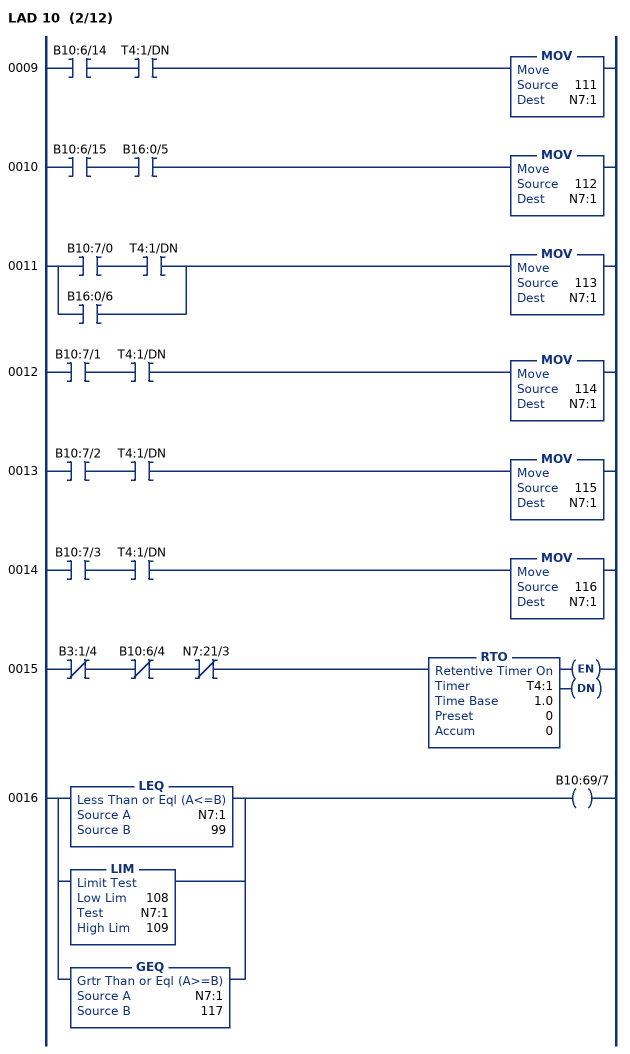
% Rung: 9 %
SOR XIC B10:6/14 XIC T4:1/DN MOV 111 N7:1 EOR
% Rung: 10 %
SOR XIC B10:6/15 XIC B16:0/5 MOV 112 N7:1 EOR
% Rung: 11 %
SOR BST XIC B10:7/0 XIC T4:1/DN NXB XIC B16:0/6 BND MOV 113 N7:1 EOR
% Rung: 12 %
SOR XIC B10:7/1 XIC T4:1/DN MOV 114 N7:1 EOR
% Rung: 13 %
SOR XIC B10:7/2 XIC T4:1/DN MOV 115 N7:1 EOR
% Rung: 14 %
SOR XIC B10:7/3 XIC T4:1/DN MOV 116 N7:1 EOR
% Rung: 15 %
SOR XIO B3:1/4 XIO B10:6/4 XIO N7:21/3 RTO T4:1 1.0 0 0 EOR
% Rung: 16 %
SOR BST LEQ N7:1 99 NXB LIM 108 N7:1 109 NXB GEQ N7:1 117 BND OTE B10:69/7 EOR

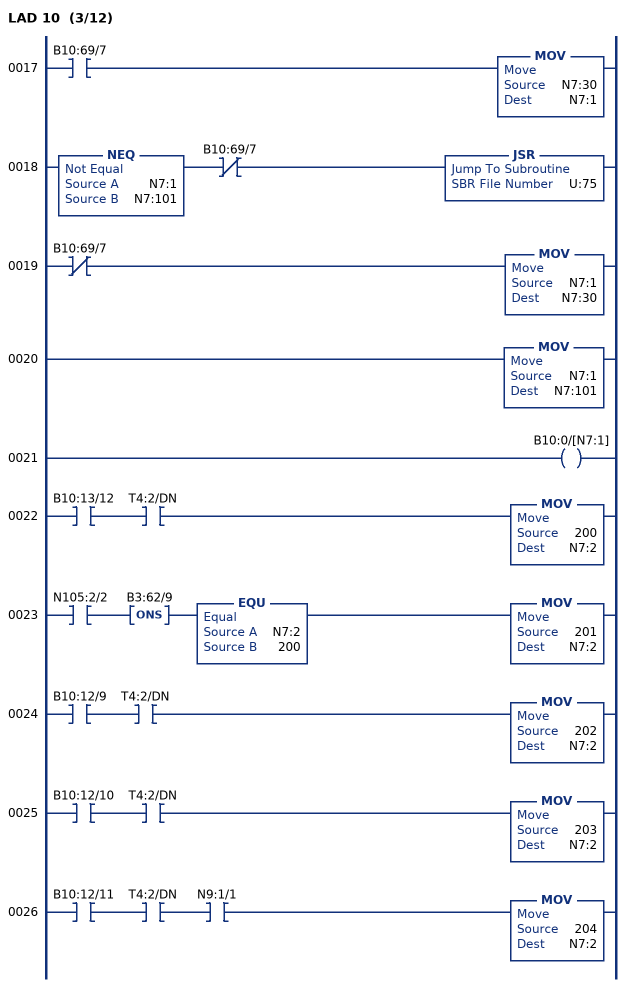
% Rung: 17 %
SOR XIC B10:69/7 MOV N7:30 N7:1 EOR
% Rung: 18 %
SOR NEQ N7:1 N7:101 XIO B10:69/7 JSR U:75 EOR
% Rung: 19 %
SOR XIO B10:69/7 MOV N7:1 N7:30 EOR
% Rung: 20 %
SOR MOV N7:1 N7:101 EOR
% Rung: 21 %
SOR OTE B10:0/[N7:1] EOR
% Rung: 22 %
SOR XIC B10:13/12 XIC T4:2/DN MOV 200 N7:2 EOR
% Rung: 23 %
SOR XIC N105:2/2 OSR B3:62/9 EQU N7:2 200 MOV 201 N7:2 EOR
% Rung: 24 %
SOR XIC B10:12/9 XIC T4:2/DN MOV 202 N7:2 EOR
% Rung: 25 %
SOR XIC B10:12/10 XIC T4:2/DN MOV 203 N7:2 EOR
% Rung: 26 %
SOR XIC B10:12/11 XIC T4:2/DN XIC N9:1/1 MOV 204 N7:2 EOR

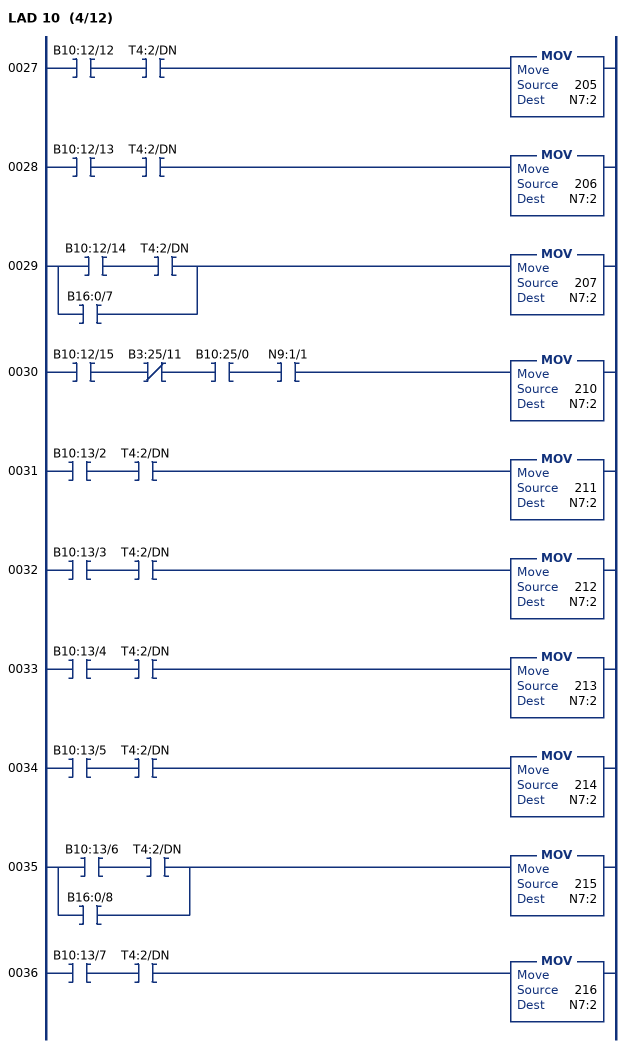
% Rung: 27 %
SOR XIC B10:12/12 XIC T4:2/DN MOV 205 N7:2 EOR
% Rung: 28 %
SOR XIC B10:12/13 XIC T4:2/DN MOV 206 N7:2 EOR
% Rung: 29 %
SOR BST XIC B10:12/14 XIC T4:2/DN NXB XIC B16:0/7 BND MOV 207 N7:2 EOR
% Rung: 30 %
SOR XIC B10:12/15 XIO B3:25/11 XIC B10:25/0 XIC N9:1/1 MOV 210 N7:2 EOR
% Rung: 31 %
SOR XIC B10:13/2 XIC T4:2/DN MOV 211 N7:2 EOR
% Rung: 32 %
SOR XIC B10:13/3 XIC T4:2/DN MOV 212 N7:2 EOR
% Rung: 33 %
SOR XIC B10:13/4 XIC T4:2/DN MOV 213 N7:2 EOR
% Rung: 34 %
SOR XIC B10:13/5 XIC T4:2/DN MOV 214 N7:2 EOR
% Rung: 35 %
SOR BST XIC B10:13/6 XIC T4:2/DN NXB XIC B16:0/8 BND MOV 215 N7:2 EOR
% Rung: 36 %
SOR XIC B10:13/7 XIC T4:2/DN MOV 216 N7:2 EOR

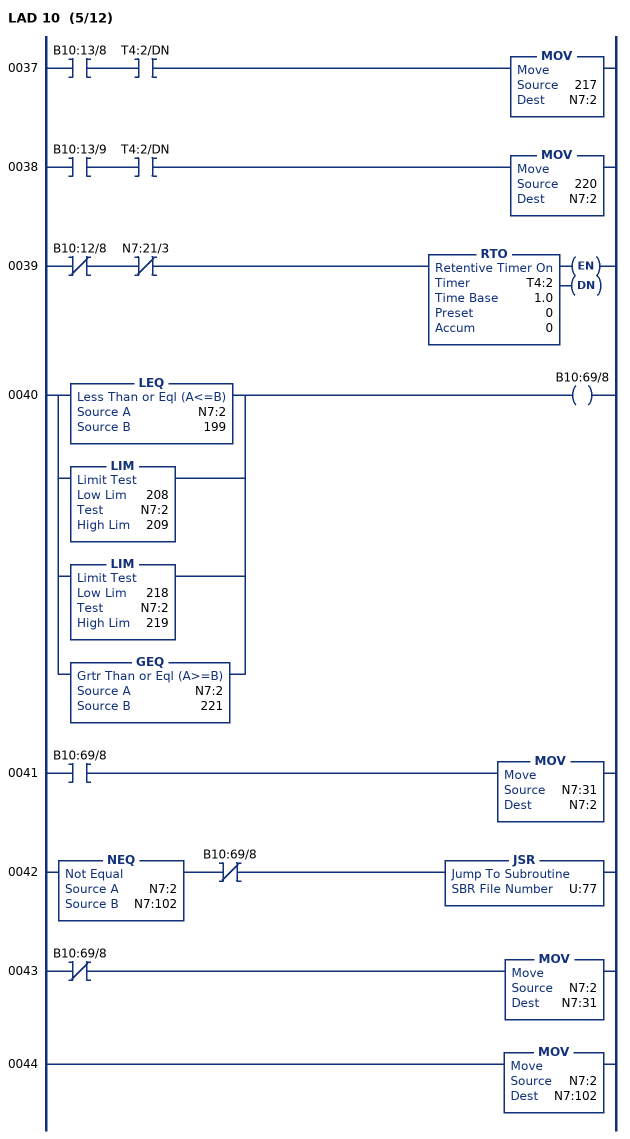
% Rung: 37 %
SOR XIC B10:13/8 XIC T4:2/DN MOV 217 N7:2 EOR
% Rung: 38 %
SOR XIC B10:13/9 XIC T4:2/DN MOV 220 N7:2 EOR
% Rung: 39 %
SOR XIO B10:12/8 XIO N7:21/3 RTO T4:2 1.0 0 0 EOR
% Rung: 40 %
SOR BST LEQ N7:2 199 NXB LIM 208 N7:2 209 NXB LIM 218 N7:2 219 NXB GEQ N7:2 221 BND OTE B10:69/8 EOR
% Rung: 41 %
SOR XIC B10:69/8 MOV N7:31 N7:2 EOR
% Rung: 42 %
SOR NEQ N7:2 N7:102 XIO B10:69/8 JSR U:77 EOR
% Rung: 43 %
SOR XIO B10:69/8 MOV N7:2 N7:31 EOR
% Rung: 44 %
SOR MOV N7:2 N7:102 EOR

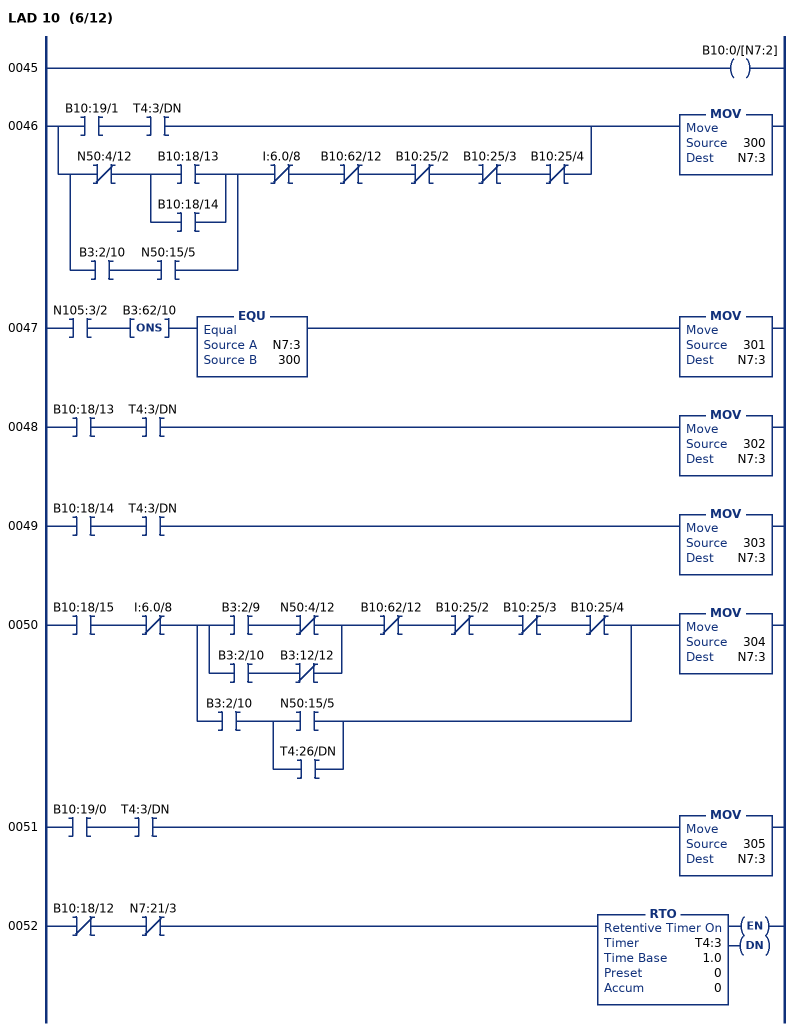
% Rung: 45 %
SOR OTE B10:0/[N7:2] EOR
% Rung: 46 %
SOR BST XIC B10:19/1 XIC T4:3/DN NXB BST XIO N50:4/12 BST XIC B10:18/13 NXB XIC B10:18/14 BND NXB XIC B3:2/10 XIC N50:15/5 BND XIO I:6.0/8 XIO B10:62/12 XIO B10:25/2 XIO B10:25/3 XIO B10:25/4 BND MOV 300 N7:3 EOR
% Rung: 47 %
SOR XIC N105:3/2 OSR B3:62/10 EQU N7:3 300 MOV 301 N7:3 EOR
% Rung: 48 %
SOR XIC B10:18/13 XIC T4:3/DN MOV 302 N7:3 EOR
% Rung: 49 %
SOR XIC B10:18/14 XIC T4:3/DN MOV 303 N7:3 EOR
% Rung: 50 %
SOR XIC B10:18/15 XIO I:6.0/8 BST BST XIC B3:2/9 XIO N50:4/12 NXB XIC B3:2/10 XIO B3:12/12 BND XIO B10:62/12 XIO B10:25/2 XIO B10:25/3 XIO B10:25/4 NXB XIC B3:2/10 BST XIC N50:15/5 NXB XIC T4:26/DN BND BND MOV 304 N7:3 EOR
% Rung: 51 %
SOR XIC B10:19/0 XIC T4:3/DN MOV 305 N7:3 EOR
% Rung: 52 %
SOR XIO B10:18/12 XIO N7:21/3 RTO T4:3 1.0 0 0 EOR

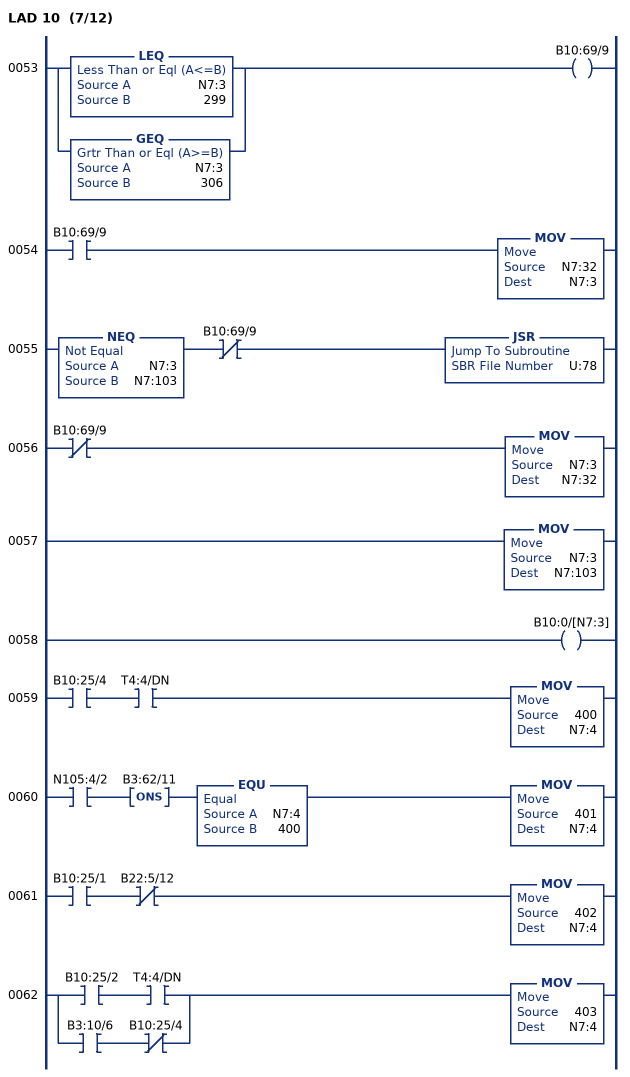
% Rung: 53 %
SOR BST LEQ N7:3 299 NXB GEQ N7:3 306 BND OTE B10:69/9 EOR
% Rung: 54 %
SOR XIC B10:69/9 MOV N7:32 N7:3 EOR
% Rung: 55 %
SOR NEQ N7:3 N7:103 XIO B10:69/9 JSR U:78 EOR
% Rung: 56 %
SOR XIO B10:69/9 MOV N7:3 N7:32 EOR
% Rung: 57 %
SOR MOV N7:3 N7:103 EOR
% Rung: 58 %
SOR OTE B10:0/[N7:3] EOR
% Rung: 59 %
SOR XIC B10:25/4 XIC T4:4/DN MOV 400 N7:4 EOR
% Rung: 60 %
SOR XIC N105:4/2 OSR B3:62/11 EQU N7:4 400 MOV 401 N7:4 EOR
% Rung: 61 %
SOR XIC B10:25/1 XIO B22:5/12 MOV 402 N7:4 EOR
% Rung: 62 %
SOR BST XIC B10:25/2 XIC T4:4/DN NXB XIC B3:10/6 XIO B10:25/4 BND MOV 403 N7:4 EOR

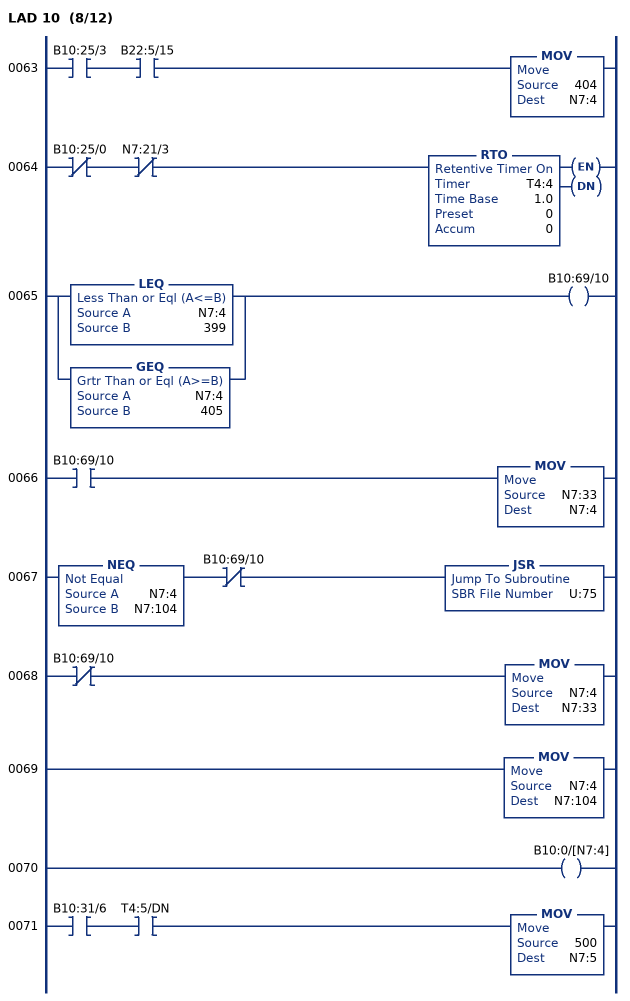
% Rung: 63 %
SOR XIC B10:25/3 XIC B22:5/15 MOV 404 N7:4 EOR
% Rung: 64 %
SOR XIO B10:25/0 XIO N7:21/3 RTO T4:4 1.0 0 0 EOR
% Rung: 65 %
SOR BST LEQ N7:4 399 NXB GEQ N7:4 405 BND OTE B10:69/10 EOR
% Rung: 66 %
SOR XIC B10:69/10 MOV N7:33 N7:4 EOR
% Rung: 67 %
SOR NEQ N7:4 N7:104 XIO B10:69/10 JSR U:75 EOR
% Rung: 68 %
SOR XIO B10:69/10 MOV N7:4 N7:33 EOR
% Rung: 69 %
SOR MOV N7:4 N7:104 EOR
% Rung: 70 %
SOR OTE B10:0/[N7:4] EOR
% Rung: 71 %
SOR XIC B10:31/6 XIC T4:5/DN MOV 500 N7:5 EOR

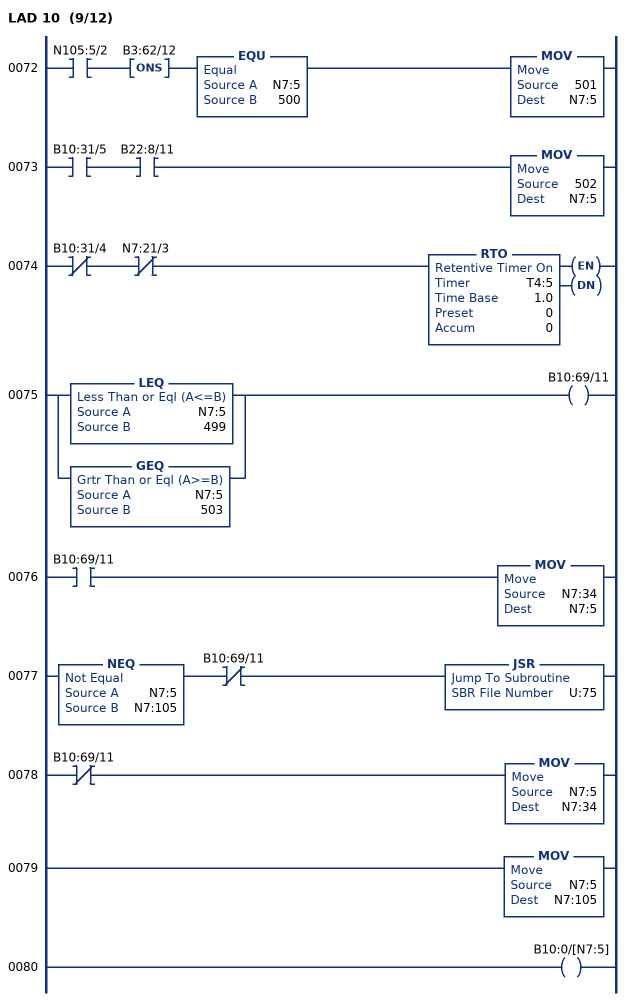
% Rung: 72 %
SOR XIC N105:5/2 OSR B3:62/12 EQU N7:5 500 MOV 501 N7:5 EOR
% Rung: 73 %
SOR XIC B10:31/5 XIC B22:8/11 MOV 502 N7:5 EOR
% Rung: 74 %
SOR XIO B10:31/4 XIO N7:21/3 RTO T4:5 1.0 0 0 EOR
% Rung: 75 %
SOR BST LEQ N7:5 499 NXB GEQ N7:5 503 BND OTE B10:69/11 EOR
% Rung: 76 %
SOR XIC B10:69/11 MOV N7:34 N7:5 EOR
% Rung: 77 %
SOR NEQ N7:5 N7:105 XIO B10:69/11 JSR U:75 EOR
% Rung: 78 %
SOR XIO B10:69/11 MOV N7:5 N7:34 EOR
% Rung: 79 %
SOR MOV N7:5 N7:105 EOR
% Rung: 80 %
SOR OTE B10:0/[N7:5] EOR

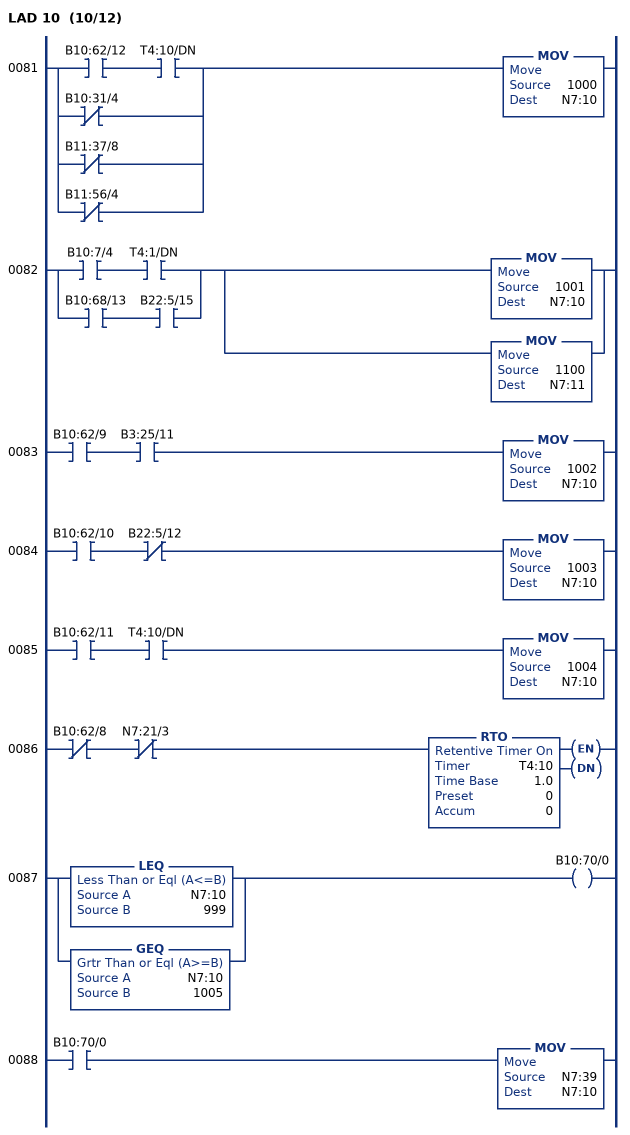
% Rung: 81 %
SOR BST XIC B10:62/12 XIC T4:10/DN NXB XIO B10:31/4 NXB XIO B11:37/8 NXB XIO B11:56/4 BND MOV 1000 N7:10 EOR
% Rung: 82 %
SOR BST XIC B10:7/4 XIC T4:1/DN NXB XIC B10:68/13 XIC B22:5/15 BND BST MOV 1001 N7:10 NXB MOV 1100 N7:11 BND EOR
% Rung: 83 %
SOR XIC B10:62/9 XIC B3:25/11 MOV 1002 N7:10 EOR
% Rung: 84 %
SOR XIC B10:62/10 XIO B22:5/12 MOV 1003 N7:10 EOR
% Rung: 85 %
SOR XIC B10:62/11 XIC T4:10/DN MOV 1004 N7:10 EOR
% Rung: 86 %
SOR XIO B10:62/8 XIO N7:21/3 RTO T4:10 1.0 0 0 EOR
% Rung: 87 %
SOR BST LEQ N7:10 999 NXB GEQ N7:10 1005 BND OTE B10:70/0 EOR
% Rung: 88 %
SOR XIC B10:70/0 MOV N7:39 N7:10 EOR

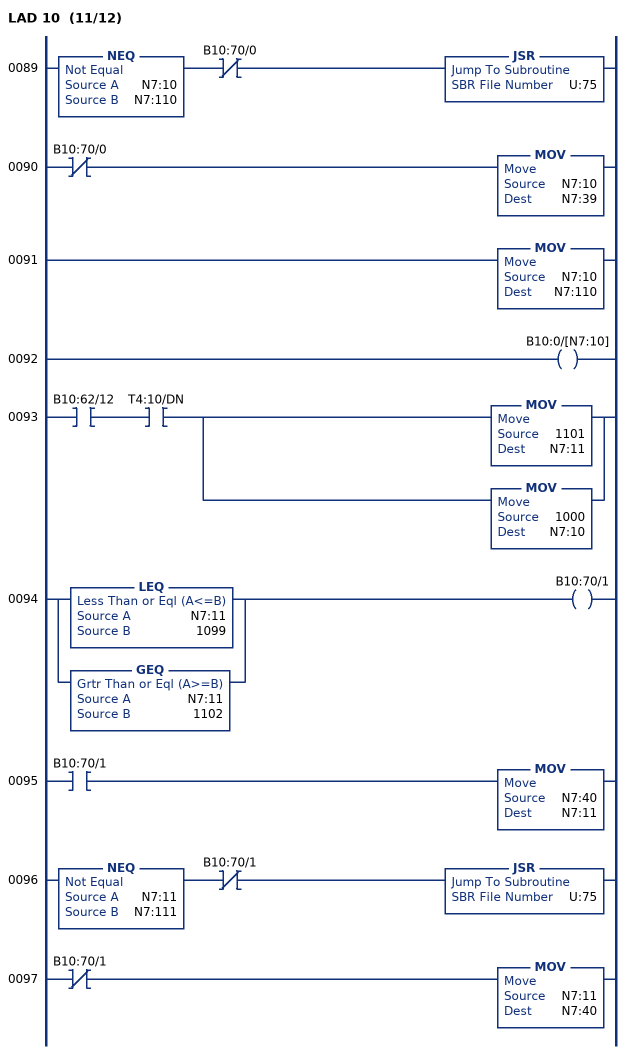
% Rung: 89 %
SOR NEQ N7:10 N7:110 XIO B10:70/0 JSR U:75 EOR
% Rung: 90 %
SOR XIO B10:70/0 MOV N7:10 N7:39 EOR
% Rung: 91 %
SOR MOV N7:10 N7:110 EOR
% Rung: 92 %
SOR OTE B10:0/[N7:10] EOR
% Rung: 93 %
SOR XIC B10:62/12 XIC T4:10/DN BST MOV 1101 N7:11 NXB MOV 1000 N7:10 BND EOR
% Rung: 94 %
SOR BST LEQ N7:11 1099 NXB GEQ N7:11 1102 BND OTE B10:70/1 EOR
% Rung: 95 %
SOR XIC B10:70/1 MOV N7:40 N7:11 EOR
% Rung: 96 %
SOR NEQ N7:11 N7:111 XIO B10:70/1 JSR U:75 EOR
% Rung: 97 %
SOR XIO B10:70/1 MOV N7:11 N7:40 EOR

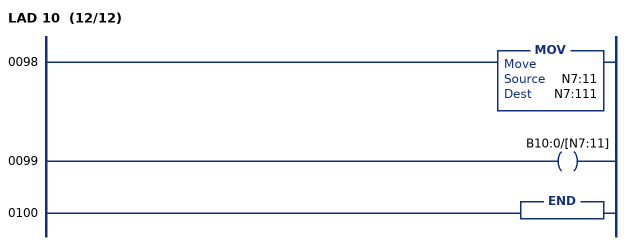
% Rung: 98 %
SOR MOV N7:11 N7:111 EOR
% Rung: 99 %
SOR OTE B10:0/[N7:11] EOR
% Rung: 100 %
SOR END EOR

LADDER 11
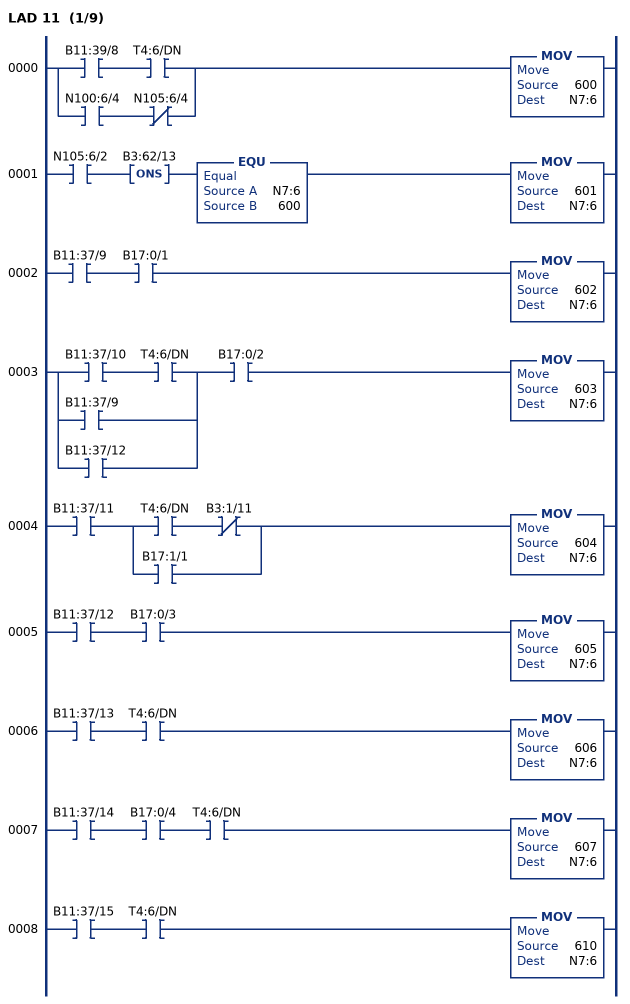
% Rung: 0 %
SOR BST XIC B11:39/8 XIC T4:6/DN NXB XIC N100:6/4 XIO N105:6/4 BND MOV 600 N7:6 EOR
% Rung: 1 %
SOR XIC N105:6/2 OSR B3:62/13 EQU N7:6 600 MOV 601 N7:6 EOR
% Rung: 2 %
SOR XIC B11:37/9 XIC B17:0/1 MOV 602 N7:6 EOR
% Rung: 3 %
SOR BST XIC B11:37/10 XIC T4:6/DN NXB BST XIC B11:37/9 NXB XIC B11:37/12 BND BND XIC B17:0/2 MOV 603 N7:6 EOR
% Rung: 4 %
SOR XIC B11:37/11 BST XIC T4:6/DN XIO B3:1/11 NXB XIC B17:1/1 BND MOV 604 N7:6 EOR
% Rung: 5 %
SOR XIC B11:37/12 XIC B17:0/3 MOV 605 N7:6 EOR
% Rung: 6 %
SOR XIC B11:37/13 XIC T4:6/DN MOV 606 N7:6 EOR
% Rung: 7 %
SOR XIC B11:37/14 XIC B17:0/4 XIC T4:6/DN MOV 607 N7:6 EOR
% Rung: 8 %
SOR XIC B11:37/15 XIC T4:6/DN MOV 610 N7:6 EOR

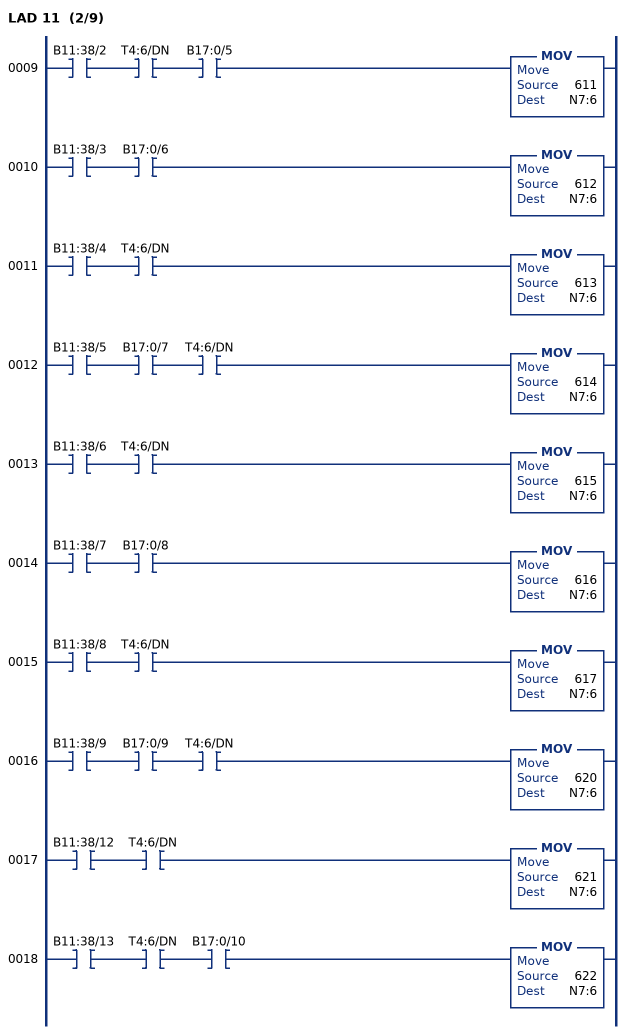
% Rung: 9 %
SOR XIC B11:38/2 XIC T4:6/DN XIC B17:0/5 MOV 611 N7:6 EOR
% Rung: 10 %
SOR XIC B11:38/3 XIC B17:0/6 MOV 612 N7:6 EOR
% Rung: 11 %
SOR XIC B11:38/4 XIC T4:6/DN MOV 613 N7:6 EOR
% Rung: 12 %
SOR XIC B11:38/5 XIC B17:0/7 XIC T4:6/DN MOV 614 N7:6 EOR
% Rung: 13 %
SOR XIC B11:38/6 XIC T4:6/DN MOV 615 N7:6 EOR
% Rung: 14 %
SOR XIC B11:38/7 XIC B17:0/8 MOV 616 N7:6 EOR
% Rung: 15 %
SOR XIC B11:38/8 XIC T4:6/DN MOV 617 N7:6 EOR
% Rung: 16 %
SOR XIC B11:38/9 XIC B17:0/9 XIC T4:6/DN MOV 620 N7:6 EOR
% Rung: 17 %
SOR XIC B11:38/12 XIC T4:6/DN MOV 621 N7:6 EOR
% Rung: 18 %
SOR XIC B11:38/13 XIC T4:6/DN XIC B17:0/10 MOV 622 N7:6 EOR

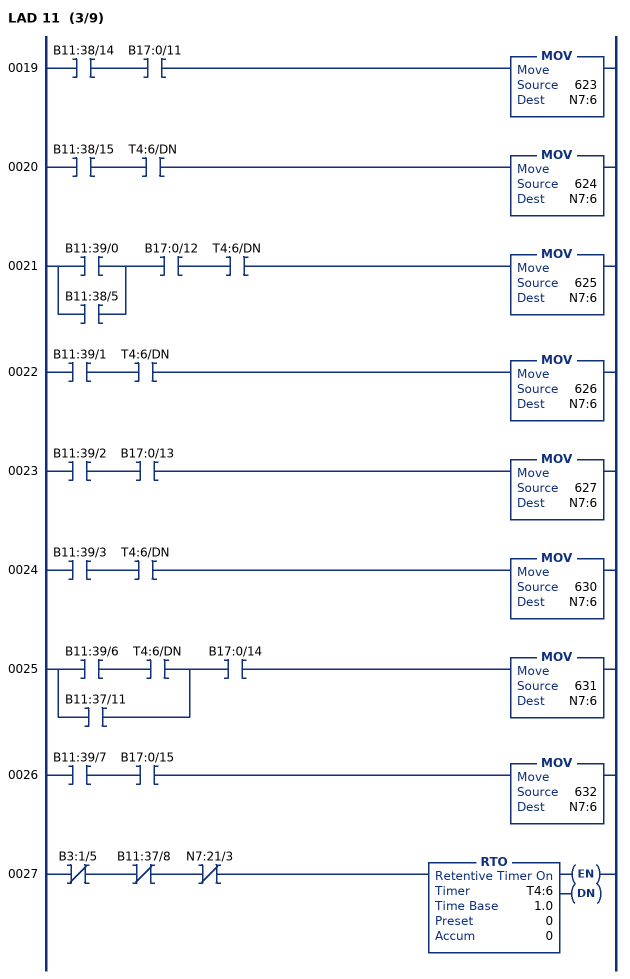
% Rung: 19 %
SOR XIC B11:38/14 XIC B17:0/11 MOV 623 N7:6 EOR
% Rung: 20 %
SOR XIC B11:38/15 XIC T4:6/DN MOV 624 N7:6 EOR
% Rung: 21 %
SOR BST XIC B11:39/0 NXB XIC B11:38/5 BND XIC B17:0/12 XIC T4:6/DN MOV 625 N7:6 EOR
% Rung: 22 %
SOR XIC B11:39/1 XIC T4:6/DN MOV 626 N7:6 EOR
% Rung: 23 %
SOR XIC B11:39/2 XIC B17:0/13 MOV 627 N7:6 EOR
% Rung: 24 %
SOR XIC B11:39/3 XIC T4:6/DN MOV 630 N7:6 EOR
% Rung: 25 %
SOR BST XIC B11:39/6 XIC T4:6/DN NXB XIC B11:37/11 BND XIC B17:0/14 MOV 631 N7:6 EOR
% Rung: 26 %
SOR XIC B11:39/7 XIC B17:0/15 MOV 632 N7:6 EOR
% Rung: 27 %
SOR XIO B3:1/5 XIO B11:37/8 XIO N7:21/3 RTO T4:6 1.0 0 0 EOR

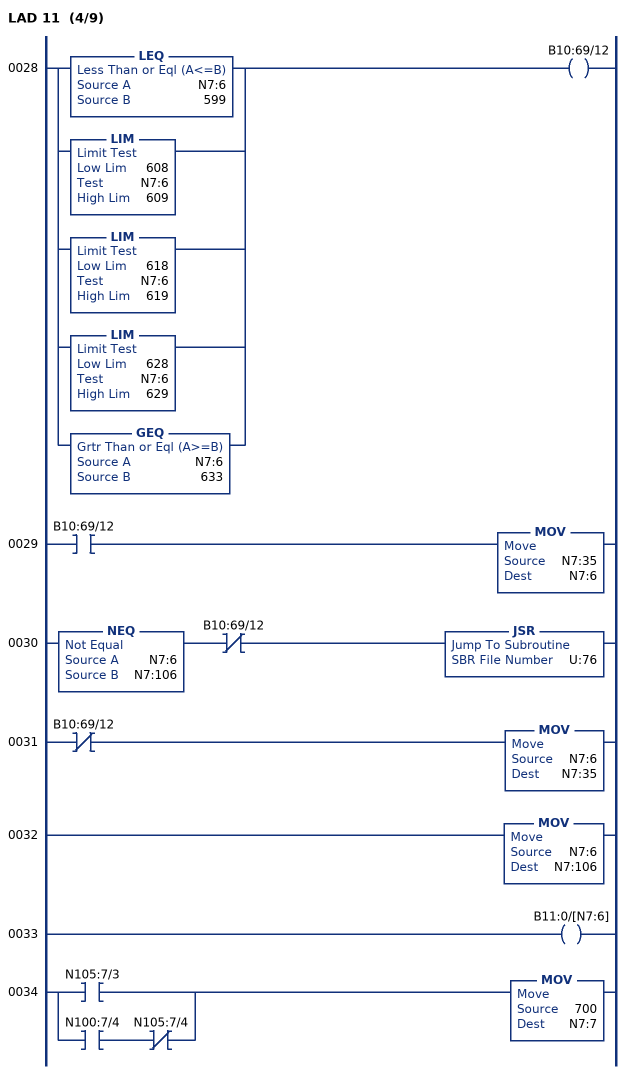
% Rung: 28 %
SOR BST LEQ N7:6 599 NXB LIM 608 N7:6 609 NXB LIM 618 N7:6 619 NXB LIM 628 N7:6 629 NXB GEQ N7:6 633 BND OTE B10:69/12 EOR
% Rung: 29 %
SOR XIC B10:69/12 MOV N7:35 N7:6 EOR
% Rung: 30 %
SOR NEQ N7:6 N7:106 XIO B10:69/12 JSR U:76 EOR
% Rung: 31 %
SOR XIO B10:69/12 MOV N7:6 N7:35 EOR
% Rung: 32 %
SOR MOV N7:6 N7:106 EOR
% Rung: 33 %
SOR OTE B11:0/[N7:6] EOR
% Rung: 34 %
SOR BST XIC N105:7/3 NXB XIC N100:7/4 XIO N105:7/4 BND MOV 700 N7:7 EOR

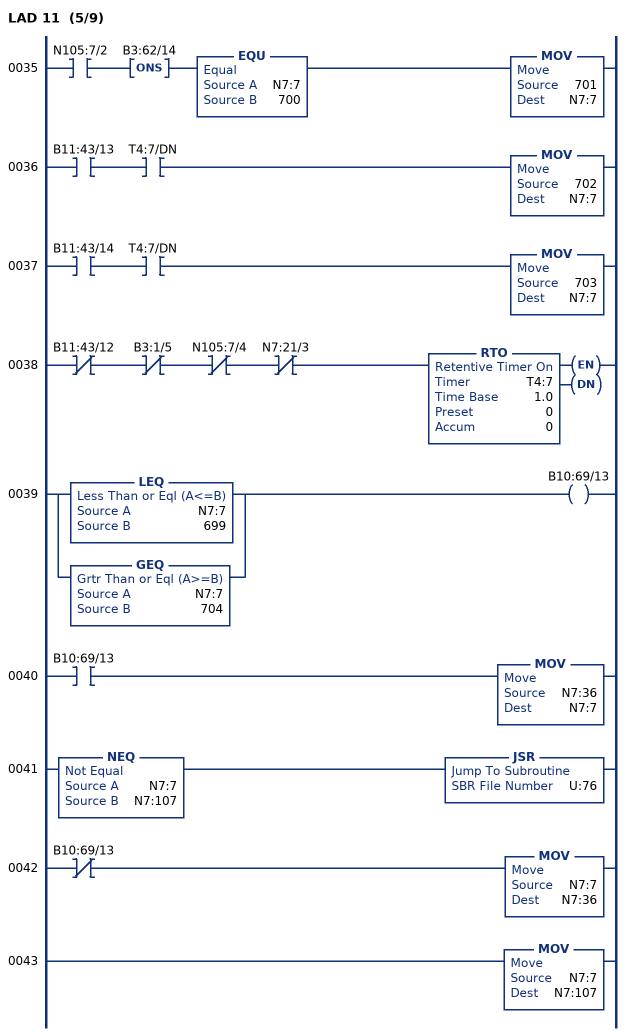
% Rung: 35 %
SOR XIC N105:7/2 OSR B3:62/14 EQU N7:7 700 MOV 701 N7:7 EOR
% Rung: 36 %
SOR XIC B11:43/13 XIC T4:7/DN MOV 702 N7:7 EOR
% Rung: 37 %
SOR XIC B11:43/14 XIC T4:7/DN MOV 703 N7:7 EOR
% Rung: 38 %
SOR XIO B11:43/12 XIO B3:1/5 XIO N105:7/4 XIO N7:21/3 RTO T4:7 1.0 0 0 EOR
% Rung: 39 %
SOR BST LEQ N7:7 699 NXB GEQ N7:7 704 BND OTE B10:69/13 EOR
% Rung: 40 %
SOR XIC B10:69/13 MOV N7:36 N7:7 EOR
% Rung: 41 %
SOR NEQ N7:7 N7:107 JSR U:76 EOR
% Rung: 42 %
SOR XIO B10:69/13 MOV N7:7 N7:36 EOR
% Rung: 43 %
SOR MOV N7:7 N7:107 EOR

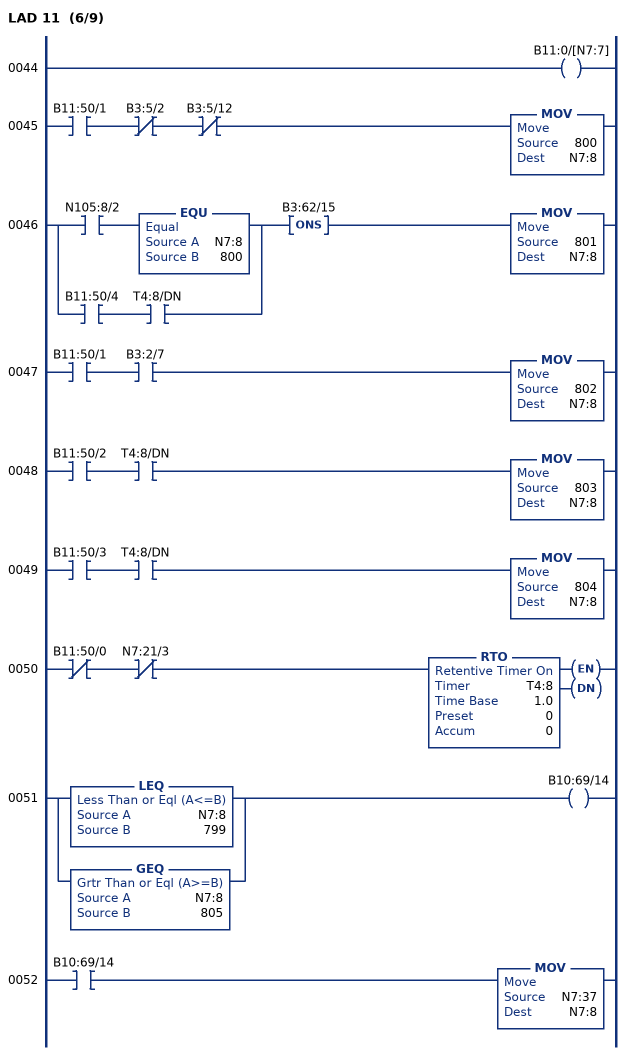
% Rung: 44 %
SOR OTE B11:0/[N7:7] EOR
% Rung: 45 %
SOR XIC B11:50/1 XIO B3:5/2 XIO B3:5/12 MOV 800 N7:8 EOR
% Rung: 46 %
SOR BST XIC N105:8/2 EQU N7:8 800 NXB XIC B11:50/4 XIC T4:8/DN BND OSR B3:62/15 MOV 801 N7:8 EOR
% Rung: 47 %
SOR XIC B11:50/1 XIC B3:2/7 MOV 802 N7:8 EOR
% Rung: 48 %
SOR XIC B11:50/2 XIC T4:8/DN MOV 803 N7:8 EOR
% Rung: 49 %
SOR XIC B11:50/3 XIC T4:8/DN MOV 804 N7:8 EOR
% Rung: 50 %
SOR XIO B11:50/0 XIO N7:21/3 RTO T4:8 1.0 0 0 EOR
% Rung: 51 %
SOR BST LEQ N7:8 799 NXB GEQ N7:8 805 BND OTE B10:69/14 EOR
% Rung: 52 %
SOR XIC B10:69/14 MOV N7:37 N7:8 EOR

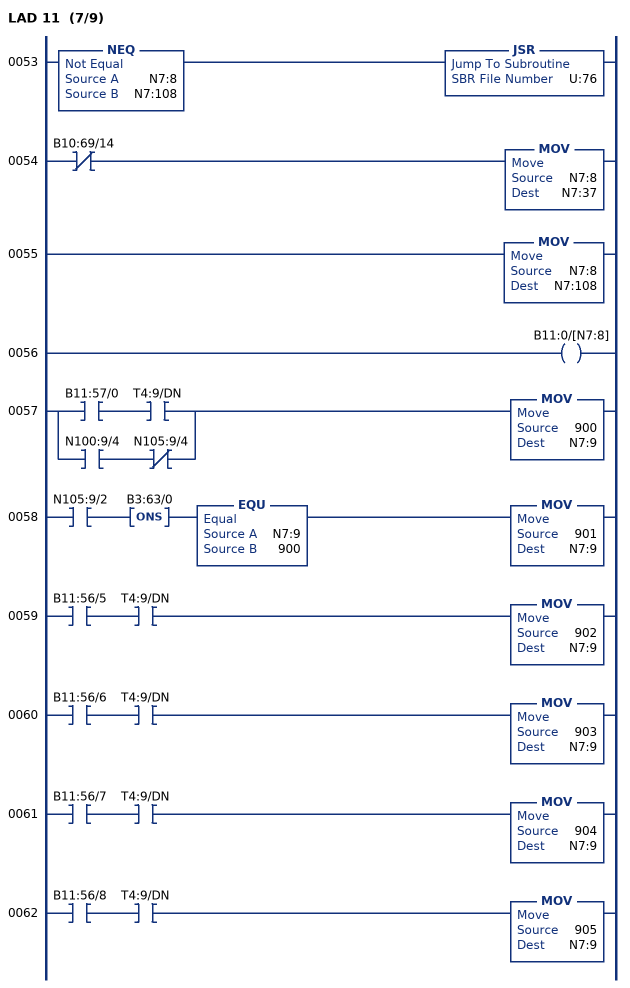
% Rung: 53 %
SOR NEQ N7:8 N7:108 JSR U:76 EOR
% Rung: 54 %
SOR XIO B10:69/14 MOV N7:8 N7:37 EOR
% Rung: 55 %
SOR MOV N7:8 N7:108 EOR
% Rung: 56 %
SOR OTE B11:0/[N7:8] EOR
% Rung: 57 %
SOR BST XIC B11:57/0 XIC T4:9/DN NXB XIC N100:9/4 XIO N105:9/4 BND MOV 900 N7:9 EOR
% Rung: 58 %
SOR XIC N105:9/2 OSR B3:63/0 EQU N7:9 900 MOV 901 N7:9 EOR
% Rung: 59 %
SOR XIC B11:56/5 XIC T4:9/DN MOV 902 N7:9 EOR
% Rung: 60 %
SOR XIC B11:56/6 XIC T4:9/DN MOV 903 N7:9 EOR
% Rung: 61 %
SOR XIC B11:56/7 XIC T4:9/DN MOV 904 N7:9 EOR
% Rung: 62 %
SOR XIC B11:56/8 XIC T4:9/DN MOV 905 N7:9 EOR

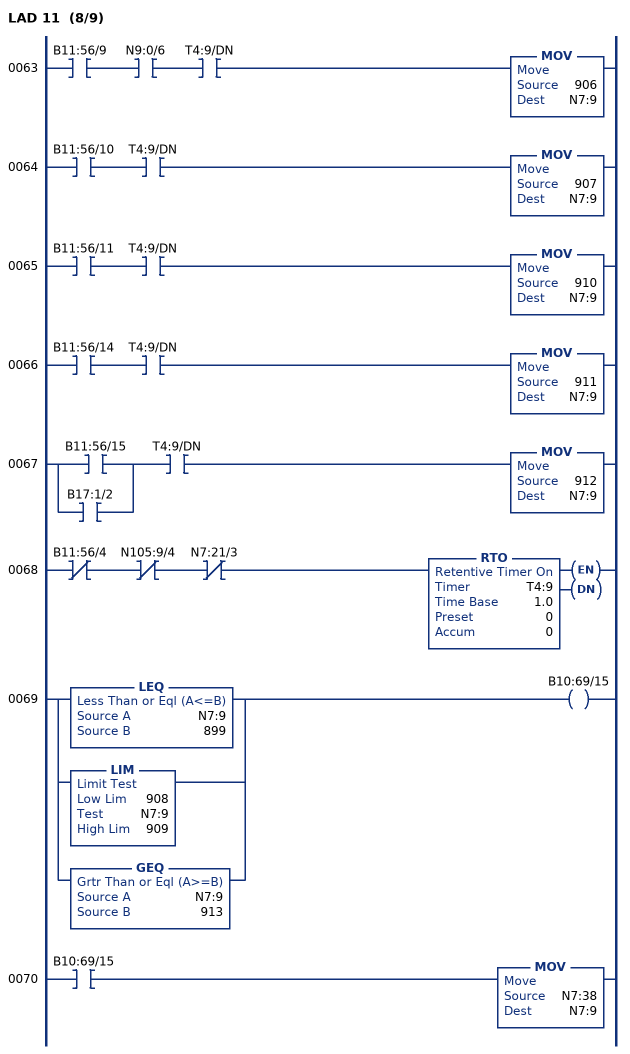
% Rung: 63 %
SOR XIC B11:56/9 XIC N9:0/6 XIC T4:9/DN MOV 906 N7:9 EOR
% Rung: 64 %
SOR XIC B11:56/10 XIC T4:9/DN MOV 907 N7:9 EOR
% Rung: 65 %
SOR XIC B11:56/11 XIC T4:9/DN MOV 910 N7:9 EOR
% Rung: 66 %
SOR XIC B11:56/14 XIC T4:9/DN MOV 911 N7:9 EOR
% Rung: 67 %
SOR BST XIC B11:56/15 NXB XIC B17:1/2 BND XIC T4:9/DN MOV 912 N7:9 EOR
% Rung: 68 %
SOR XIO B11:56/4 XIO N105:9/4 XIO N7:21/3 RTO T4:9 1.0 0 0 EOR
% Rung: 69 %
SOR BST LEQ N7:9 899 NXB LIM 908 N7:9 909 NXB GEQ N7:9 913 BND OTE B10:69/15 EOR
% Rung: 70 %
SOR XIC B10:69/15 MOV N7:38 N7:9 EOR

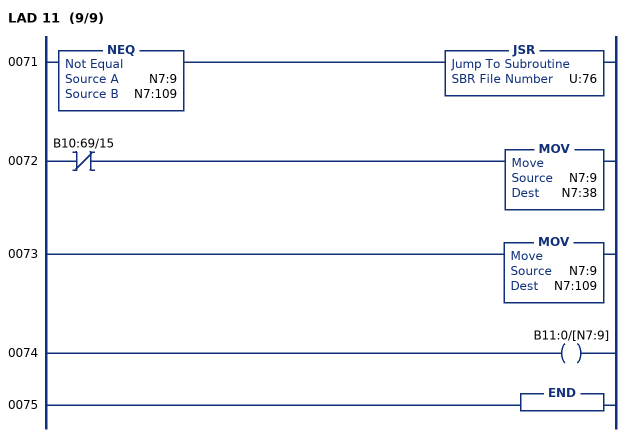
% Rung: 71 %
SOR NEQ N7:9 N7:109 JSR U:76 EOR
% Rung: 72 %
SOR XIO B10:69/15 MOV N7:9 N7:38 EOR
% Rung: 73 %
SOR MOV N7:9 N7:109 EOR
% Rung: 74 %
SOR OTE B11:0/[N7:9] EOR
% Rung: 75 %
SOR END EOR

LADDER 15
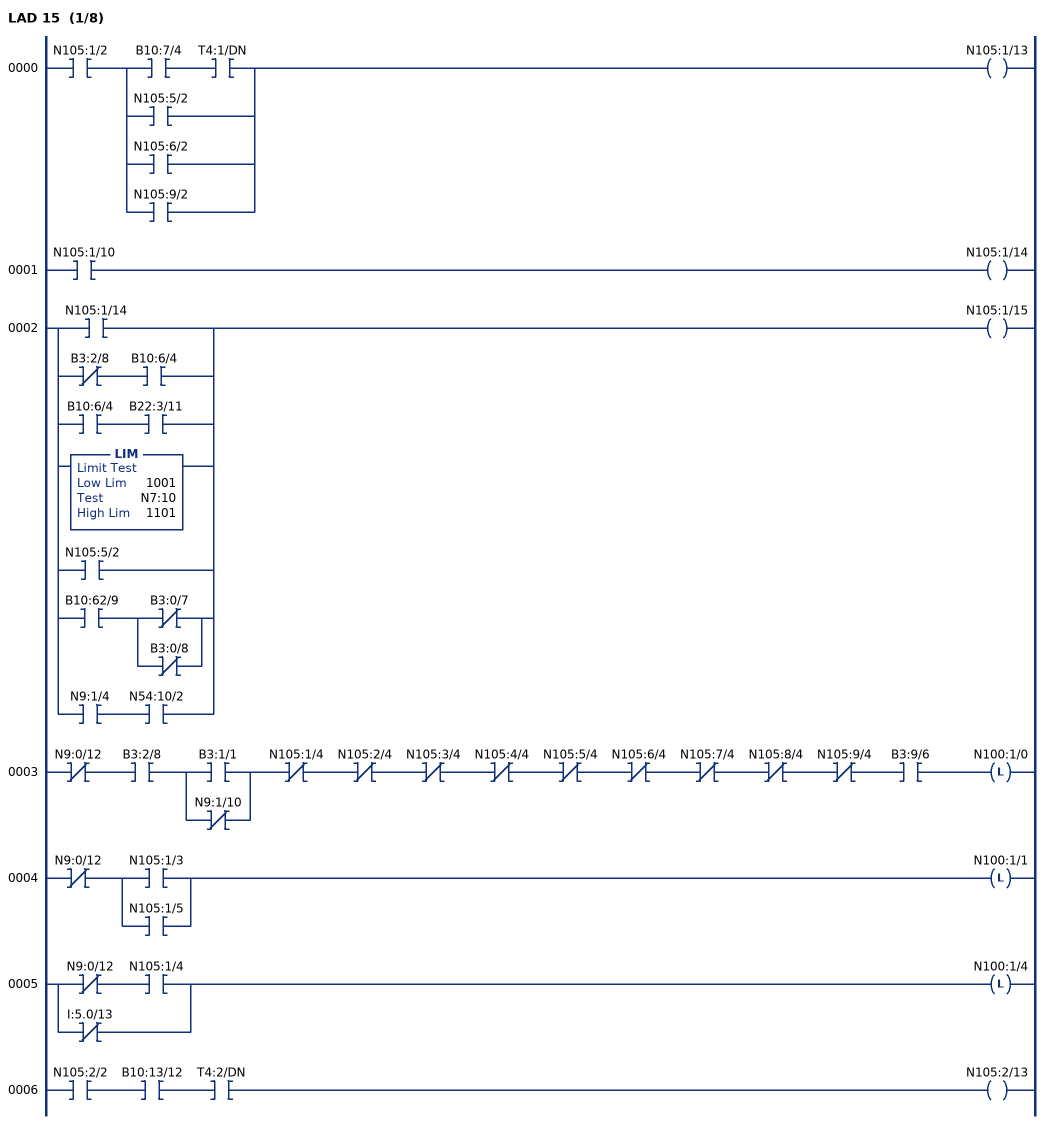
% Rung: 0 %
SOR XIC N105:1/2 BST XIC B10:7/4 XIC T4:1/DN NXB XIC N105:5/2 NXB XIC N105:6/2 NXB XIC N105:9/2 BND OTE N105:1/13 EOR
% Rung: 1 %
SOR XIC N105:1/10 OTE N105:1/14 EOR
% Rung: 2 %
SOR BST XIC N105:1/14 NXB XIO B3:2/8 XIC B10:6/4 NXB XIC B10:6/4 XIC B22:3/11 NXB LIM 1001 N7:10 1101 NXB XIC N105:5/2 NXB XIC B10:62/9 BST XIO B3:0/7 NXB XIO B3:0/8 BND NXB XIC N9:1/4 XIC N54:10/2 BND OTE N105:1/15 EOR
% Rung: 3 %
SOR XIO N9:0/12 XIC B3:2/8 BST XIC B3:1/1 NXB XIO N9:1/10 BND XIO N105:1/4 XIO N105:2/4 XIO N105:3/4 XIO N105:4/4 XIO N105:5/4 XIO N105:6/4 XIO N105:7/4 XIO N105:8/4 XIO N105:9/4 XIC B3:9/6 OTL N100:1/0 EOR
% Rung: 4 %
SOR XIO N9:0/12 BST XIC N105:1/3 NXB XIC N105:1/5 BND OTL N100:1/1 EOR
% Rung: 5 %
SOR BST XIO N9:0/12 XIC N105:1/4 NXB XIO I:5.0/13 BND OTL N100:1/4 EOR
% Rung: 6 %
SOR XIC N105:2/2 XIC B10:13/12 XIC T4:2/DN OTE N105:2/13 EOR

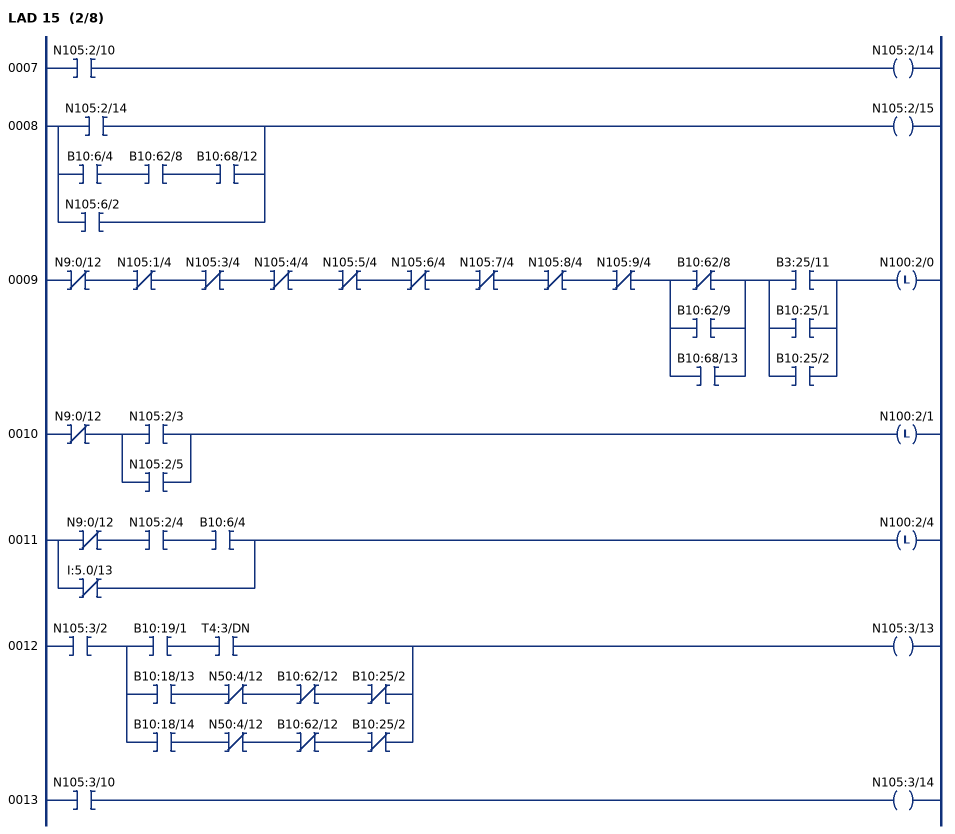
% Rung: 7 %
SOR XIC N105:2/10 OTE N105:2/14 EOR
% Rung: 8 %
SOR BST XIC N105:2/14 NXB XIC B10:6/4 XIC B10:62/8 XIC B10:68/12 NXB XIC N105:6/2 BND OTE N105:2/15 EOR
% Rung: 9 %
SOR XIO N9:0/12 XIO N105:1/4 XIO N105:3/4 XIO N105:4/4 XIO N105:5/4 XIO N105:6/4 XIO N105:7/4 XIO N105:8/4 XIO N105:9/4 BST XIO B10:62/8 NXB XIC B10:62/9 NXB XIC B10:68/13 BND BST XIC B3:25/11 NXB XIC B10:25/1 NXB XIC B10:25/2 BND OTL N100:2/0 EOR
% Rung: 10 %
SOR XIO N9:0/12 BST XIC N105:2/3 NXB XIC N105:2/5 BND OTL N100:2/1 EOR
% Rung: 11 %
SOR BST XIO N9:0/12 XIC N105:2/4 XIC B10:6/4 NXB XIO I:5.0/13 BND OTL N100:2/4 EOR
% Rung: 12 %
SOR XIC N105:3/2 BST XIC B10:19/1 XIC T4:3/DN NXB XIC B10:18/13 XIO N50:4/12 XIO B10:62/12 XIO B10:25/2 NXB XIC B10:18/14 XIO N50:4/12 XIO B10:62/12 XIO B10:25/2 BND OTE N105:3/13 EOR
% Rung: 13 %
SOR XIC N105:3/10 OTE N105:3/14 EOR

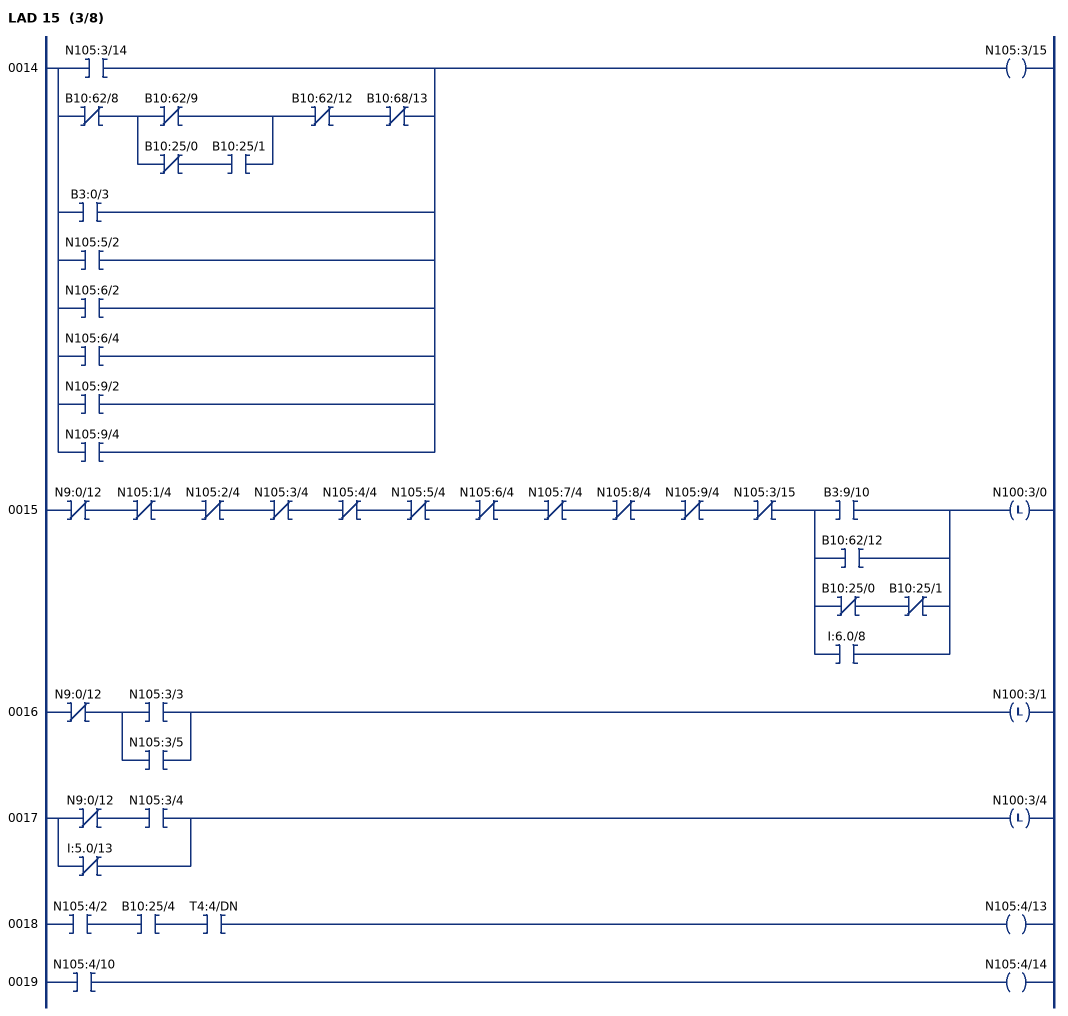
% Rung: 14 %
SOR BST XIC N105:3/14 NXB XIO B10:62/8 BST XIO B10:62/9 NXB XIO B10:25/0 XIC B10:25/1 BND XIO B10:62/12 XIO B10:68/13 NXB XIC B3:0/3 NXB XIC N105:5/2 NXB XIC N105:6/2 NXB XIC N105:6/4 NXB XIC N105:9/2 NXB XIC N105:9/4 BND OTE N105:3/15 EOR
% Rung: 15 %
SOR XIO N9:0/12 XIO N105:1/4 XIO N105:2/4 XIO N105:3/4 XIO N105:4/4 XIO N105:5/4 XIO N105:6/4 XIO N105:7/4 XIO N105:8/4 XIO N105:9/4 XIO N105:3/15 BST XIC B3:9/10 NXB XIC B10:62/12 NXB XIO B10:25/0 XIO B10:25/1 NXB XIC I:6.0/8 BND OTL N100:3/0 EOR
% Rung: 16 %
SOR XIO N9:0/12 BST XIC N105:3/3 NXB XIC N105:3/5 BND OTL N100:3/1 EOR
% Rung: 17 %
SOR BST XIO N9:0/12 XIC N105:3/4 NXB XIO I:5.0/13 BND OTL N100:3/4 EOR
% Rung: 18 %
SOR XIC N105:4/2 XIC B10:25/4 XIC T4:4/DN OTE N105:4/13 EOR
% Rung: 19 %
SOR XIC N105:4/10 OTE N105:4/14 EOR

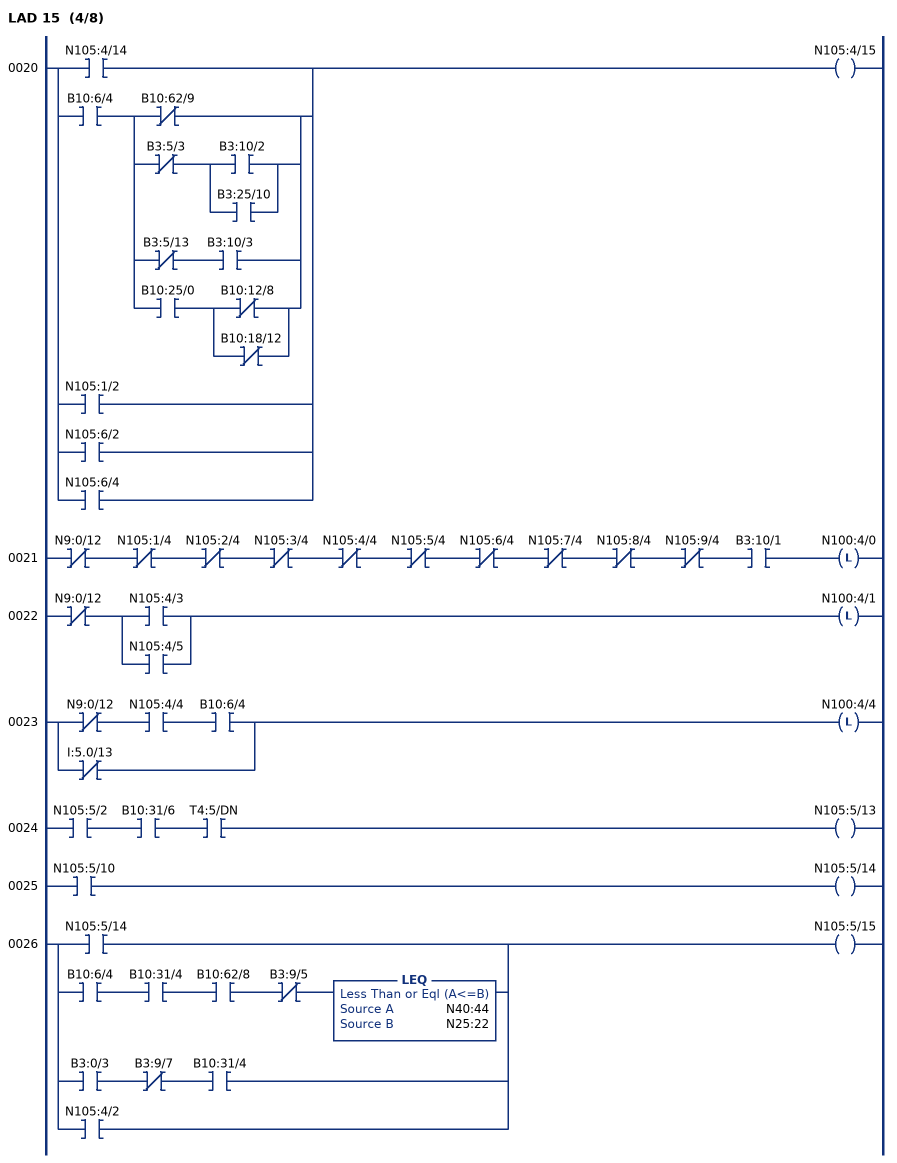
% Rung: 20 %
SOR BST XIC N105:4/14 NXB XIC B10:6/4 BST XIO B10:62/9 NXB XIO B3:5/3 BST XIC B3:10/2 NXB XIC B3:25/10 BND NXB XIO B3:5/13 XIC B3:10/3 NXB XIC B10:25/0 BST XIO B10:12/8 NXB XIO B10:18/12 BND BND NXB XIC N105:1/2 NXB XIC N105:6/2 NXB XIC N105:6/4 BND OTE N105:4/15 EOR
% Rung: 21 %
SOR XIO N9:0/12 XIO N105:1/4 XIO N105:2/4 XIO N105:3/4 XIO N105:4/4 XIO N105:5/4 XIO N105:6/4 XIO N105:7/4 XIO N105:8/4 XIO N105:9/4 XIC B3:10/1 OTL N100:4/0 EOR
% Rung: 22 %
SOR XIO N9:0/12 BST XIC N105:4/3 NXB XIC N105:4/5 BND OTL N100:4/1 EOR
% Rung: 23 %
SOR BST XIO N9:0/12 XIC N105:4/4 XIC B10:6/4 NXB XIO I:5.0/13 BND OTL N100:4/4 EOR
% Rung: 24 %
SOR XIC N105:5/2 XIC B10:31/6 XIC T4:5/DN OTE N105:5/13 EOR
% Rung: 25 %
SOR XIC N105:5/10 OTE N105:5/14 EOR
% Rung: 26 %
SOR BST XIC N105:5/14 NXB XIC B10:6/4 XIC B10:31/4 XIC B10:62/8 XIO B3:9/5 LEQ N40:44 N25:22 NXB XIC B3:0/3 XIO B3:9/7 XIC B10:31/4 NXB XIC N105:4/2 BND OTE N105:5/15 EOR

